PROGRAM DomeControl
VAR_INPUT
	// enable the dome azimuth
	enable:		BOOL;
	// reset the dome axis after an error
	Reset:		BOOL;
	// rotate the dome left (ccw)
	left:		BOOL;
	// rotate the dome right (cw)
	right: 		BOOL;
	// open the dome
	OpenDome:	BOOL;
	// close the dome
	CloseDome:	BOOL; // := TRUE;
	// turn on the light in the dome
	Light: 		BOOL;
	// azimuth position to move to
	position:	LREAL;
	// initiate homing
	HomeAxis:	BOOL;
END_VAR
VAR_OUTPUT
	// error condition on the azimuth drive
	Error:		BOOL;
	// NC axis error of the dome drive
	ErrorID:	UDINT;
	// error in the dome communication or drive
	DomeError:	BOOL;
	// dome is calibrated
	Calibrated:	BOOL;
END_VAR
VAR
	// dome axis function block
	DomeAxis: FB_Axis2;
	// current measured dome azimuth
	Azimuth_current: 	LREAL;
	// dome velocity
	ActVelo:			LREAL;
	//
	//manual_enable:		BOOL;
	// command to move the azimuth to position
	move_azimuth:		BOOL;
	// dome is halted
	//stop_done:			BOOL;
	// dome slit and flap are open
	DomeOpened:			BOOL;
	// dome is closed
	DomeClosed:			BOOL;
	// dome flap (lower section) is open
	FlapOpen:			BOOL;
	// dome flap (lower section) is closed
	FlapClosed:			BOOL;
	//dome slit is open
	SlitOpen:			BOOL;
	// dome slit is closed
	SlitClosed:			BOOL;
	// bit to indicate if domestatus is valid
	DomeValid:			BOOL;
	// dome control word
   	DomeStatusWord:		WORD;
	// last status Word
	LastStatus:			WORD;
	// permanent communication error
	PermanentError:		TON := (IN:=FALSE, PT:=T#30S);
	HomeDelay:			FB_TONTP;
	F_Azimuth_home:		F_TRIG;
	R_Azimuth_home:		R_TRIG;
	// direction invariant azimuth home signal;
	Azimuth_home:		BOOL;
	// time delay for dome light
	LightTimer:			TP;
	// next state
	//:				BYTE := 0;
	// ADS communiaction busy
	bBusy: 				BOOL;
	// ADS communication error
	bError: 			BOOL;
	// ADS communication error id
	nErrID: 			UDINT;
	// cycle timer for the ADS write cycle
	ReadCycle:			TON := (PT:=T#1S);
	
	fbReadReq: ADSREAD := ( NETID := '5.73.45.158.1.1', PORT := 851, TMOUT := DEFAULT_ADS_TIMEOUT );
	DomeCalibration:	MC_SetPosition;
	SyncDome:			BOOL;
	DomeCommEvent:		FB_Eventlog;
	DomeAxisEvent:		FB_Eventlog;
	DomeOpenedEvent:	FB_Eventlog;
	DomeClosedEvent:	FB_Eventlog;
	OpenDomeEvent:		FB_Eventlog;
	CloseDomeEvent:		FB_Eventlog;
	DomeCalibrationEvent: FB_Eventlog;
	MQTTTimer : TON := (PT:=T#10S);
	// MQTT String
	sPayloadPub: STRING(255);
	getlastposition:	BOOL := TRUE;
END_VAR
VAR CONSTANT
	tolerance:				LREAL := 5.0;
	calibration_position:	LREAL := 172.5;
	home_position:			LREAL := 180.0;
END_VAR
VAR PERSISTENT
	last_position:	LREAL := -1.0;
END_VAR

(* This program is responsible for the dome control. 
The dome is enabled unless the emergency button is pressed.
The two-button manual box steers the dome counter-clockwise or clockwise
If the dome is in automatic mode, homing is performed first.
The first section controls the signals for the inverter.
The second section controls the dome axis.
The third section handles the communications via ADS with the dome PLC.
*)

DomeLowLevelControl(enable := GVL_Safety.Run);
enable := GVL_Safety.Run;

// if we are calibrated or encounter an error while calibrating, deactivate homing
IF DomeAxis.Calibrated OR Error THEN
	HomeAxis := FALSE;
END_IF

IF Error THEN
	move_azimuth := FALSE;
END_IF

IF DomeAxis.Calibrated THEN
	last_position := Azimuth_current;
	getlastposition := FALSE;
END_IF


ActVelo := GVL_Dome.ActVelo;

// limit position to sane value
position := MODABS(position, 360.0);

// if we are calibrated, but azimuth is not, go to home position
HomeDelay(IN := DomeAxis.Calibrated, PT1 := T#5S, PT2 := T#100MS);

IF HomeDelay.Q THEN
	position := home_position;
	move_azimuth := TRUE;
END_IF

SyncDome := DomeAxis.Calibrated AND TelescopeControl.power AND AzimuthElevationControl.calibrated;
// if we are on automatic, tie the dome to the telescope

IF DomeAxis.Calibrated AND TelescopeControl.power AND AzimuthElevationControl.calibrated THEN
	position := MODABS(TelescopeControl.azimuth_current, 360.0);
	IF ABS(Azimuth_current - position) > tolerance THEN
		move_azimuth := TRUE;
	ELSE
		move_azimuth := FALSE;
	END_IF
	
END_IF

Calibrated := DomeAxis.Calibrated;
// when homing, ensure that the position is the calibration position
IF HomeAxis THEN
	position := calibration_position;	
END_IF
F_Azimuth_home(CLK := GVL_Dome.Azimut_home);
R_Azimuth_home(CLK := GVL_Dome.Azimut_home);

Azimuth_home := (R_Azimuth_home.Q AND GVL_Dome.bDirectionPlus) OR 
				(F_Azimuth_home.Q AND GVL_Dome.bDirectionMinus);

// velocity = 2°/s or 180° in 81s, 360° in 120s (was 2.22)
// TODO: Reset does not propagate to the FB and therefor does not reset the error
DomeAxis(
	Enable := 		enable,
	Reset := 		reset,
	MoveAxis := 	move_azimuth,
	HomeAxis :=		HomeAxis,
	Position := 	position,
	Velocity := 	3.0,
	Jog_Forward :=	right OR GVL_Dome.Clockwise,
	Jog_Backwards := left OR GVL_Dome.CounterClockwise,
	bCalibrationCam := GVL_Dome.Azimut_home,
	isModuloAxis := TRUE,
	//StopDone =>		stop_done,
	Error =>		error,
	ErrorID =>		ErrorID,
	ActualPosition => Azimuth_current,
	AxisRef	:= 		GVL_Dome.DomeAxisRef);

IF getlastposition AND last_position>=0.0 AND NOT Calibrated THEN
	DomeCalibration.Execute := getlastposition AND DomeAxis.Ready;
	DomeCalibration.Position := last_position;
ELSE
	DomeCalibration.Execute := Azimuth_home AND HomeDelay.Q AND DomeAxis.Ready;
	DomeCalibration.Position := calibration_position;
END_IF

// re-calibrate the dome, if we pass the reference switch. execute only if enough time has passed since homing.
DomeCalibration(Axis := GVL_Dome.DomeAxisRef);

IF DomeCalibration.Done OR Calibrated THEN
	getlastposition := FALSE;
END_IF

IF DomeAxis.MoveDone THEN
	move_azimuth := FALSE;
END_IF


// Light is switched off after 60 minutes or if Light signal is low
LightTimer(IN := Light, PT := T#60M);
GVL_Dome.Light := Light AND LightTimer.Q;

(* The remote section for moving parts of the dome starts here. *)
GVL_Dome.DomeControlWord.0 := TRUE;
IF CloseDome THEN
	OpenDome := FALSE;
	GVL_Dome.DomeControlWord.1 := TRUE; // CloseFlap
	GVL_Dome.DomeControlWord.2 := TRUE; // CloseSlit
	GVL_Dome.DomeControlWord.3 := FALSE; // OpenFlap
	GVL_Dome.DomeControlWord.4 := FALSE; // OpenSlit
ELSIF OpenDome THEN
	GVL_Dome.DomeControlWord.1 := FALSE; // CloseFlap
	GVL_Dome.DomeControlWord.2 := FALSE; // CloseSlit
	GVL_Dome.DomeControlWord.3 := TRUE; // OpenFlap
	GVL_Dome.DomeControlWord.4 := TRUE; // OpenSlit
ELSE
	GVL_Dome.DomeControlWord.1 := FALSE; // CloseFlap
	GVL_Dome.DomeControlWord.2 := FALSE; // CloseSlit
	GVL_Dome.DomeControlWord.3 := FALSE; // OpenFlap
	GVL_Dome.DomeControlWord.4 := FALSE; // OpenSlit
END_IF

ReadCycle(IN := TRUE);
IF ReadCycle.Q THEN
	// read if the ADS command is busy
	fbReadReq(	READ := FALSE,
				BUSY => bBusy,
				ERR =>	bError,
				ERRID => nErrID);
	IF bBusy THEN
		// reset the read command
		fbReadReq(READ := FALSE);
	ELSE
		// read the variable
		fbReadReq(  IDXGRP := 16#4020, 
					IDXOFFS := 0, 
					LEN := SIZEOF(DomeStatusWord), 
					DESTADDR := ADR(DomeStatusWord),
					READ := TRUE,
					BUSY => bBusy,
					ERR =>	bError,
					ERRID => nErrID);
		// restart the read cycle
		ReadCycle(IN := FALSE);		
	END_IF
	
	IF NOT bError THEN
		DomeValid  := DomeStatusWord.0;
		DomeOpened := DomeStatusWord.1;
		DomeClosed := DomeStatusWord.2;
		FlapOpen   := DomeStatusWord.3;
		FlapClosed := DomeStatusWord.4;
		SlitOpen   := DomeStatusWord.5;
		SlitClosed := DomeStatusWord.6;
	ELSE
		// reset the status word
		DomeStatusWord := 0;
	END_IF
END_IF

CASE NErrID OF
			6: DomeCommEvent.OnMessage := 'ERR_TARGETPORTNOTFOUND';
			29: DomeCommEvent.OnMessage := 'ERR_AMSSYNC_TIMEOUT';
			1861: DomeCommEvent.OnMessage := 'ADSERR_CLIENT_SYNCTIMEOUT';
ELSE
			DomeCommEvent.OnMessage := UDINT_TO_STRING(nErrID);
END_CASE

PermanentError(IN := bError);
		
DomeError := PermanentError.Q OR Error;

IF DomeOpened THEN
	OpenDome := FALSE;
ELSIF DomeClosed THEN
	CloseDome := FALSE;
END_IF

MQTTTimer(IN:=Enable);
IF MQTTTimer.Q THEN // publish new payload every second
	MQTTTimer(IN:=FALSE);
	sPayloadPub := 'dome,location=dome,host=CX-4E6032 ';
	sPayloadPub := APPEND(sPayloadPub, 'DomeAzimuth=', LREAL_TO_FMTSTR(Azimuth_current, 1, TRUE));
	sPayloadPub := APPEND(sPayloadPub, ',Calibrated=', BOOL_TO_STRING(Calibrated));	
	MQTTCommunication.fbMqttClient.Publish(	
					sTopic:= 'RoboTel/Telemetry', 
					pPayload:= ADR(sPayloadPub), 
					nPayloadSize:= LEN2(ADR(sPayloadPub)),
					eQoS:= TcIotMqttQos.AtMostOnceDelivery,
					bRetain:= FALSE, 
					bQueue:= FALSE );
	// invalidate last status for testing
	LastStatus := 0;
END_IF

IF DomeStatusWord <> LastStatus THEN
	LastStatus := DomeStatusWord;
	sPayloadPub := 'dome,location=dome,host=CX-4E6032,module=DomeControl ';
	sPayloadPub := APPEND(sPayloadPub, 'DomeCommunicationOK=', BOOL_TO_STRING(NOT PermanentError.Q));
	sPayloadPub := APPEND(sPayloadPub, ',DomeClosed=', BOOL_TO_STRING(DomeClosed));
	sPayloadPub := APPEND(sPayloadPub, ',DomeOpened=', BOOL_TO_STRING(DomeOpened));
	sPayloadPub := APPEND(sPayloadPub, ',FlapOpen=', BOOL_TO_STRING(FlapOpen));	
	sPayloadPub := APPEND(sPayloadPub, ',FlapClosed=', BOOL_TO_STRING(FlapClosed));	
	sPayloadPub := APPEND(sPayloadPub, ',SlitOpen=', BOOL_TO_STRING(SlitOpen));	
	sPayloadPub := APPEND(sPayloadPub, ',SlitClosed=', BOOL_TO_STRING(SlitClosed));	
	
	MQTTCommunication.fbMqttClient.Publish(	
					sTopic:= 'RoboTel/Telemetry', 
					pPayload:= ADR(sPayloadPub), 
					nPayloadSize:= LEN2(ADR(sPayloadPub)),
					eQoS:= TcIotMqttQos.AtMostOnceDelivery,
					bRetain:= TRUE, 
					bQueue:= FALSE );
END_IF

DomeCommEvent(	Trigger := PermanentError.Q, 
					Level := ADSLOG_MSGTYPE_ERROR,
					FormatString := 'Dome communication error: %s',
					OffMessage := 'OK',
					OffLevel := ADSLOG_MSGTYPE_HINT);
DomeAxisEvent(	
	Trigger := 		Error, 
	Level := 		ADSLOG_MSGTYPE_ERROR,
	FormatString :=	'Dome axis Error: %s',
	OnMessage := 	NCError_TO_STRING(ErrorID),
	OffMEssage := 	'OK');
				
DomeCalibrationEvent(	
	Trigger := 		GVL_Dome.Azimut_home, 
	Level := 		ADSLOG_MSGTYPE_HINT,
	OnMessage := 	'Dome is (re-)calibrated.');

DomeOpenedEvent(
	Trigger := 		DomeOpened, 
	Level := 		ADSLOG_MSGTYPE_WARN,
	OnMessage := 	'Dome is open.');
	
DomeClosedEvent(
	Trigger := 		DomeClosed, 
	Level := 		ADSLOG_MSGTYPE_HINT,
	OnMessage := 	'Dome is closed.');
	
OpenDomeEvent(
	Trigger := 		OpenDome, 
	Level := 		ADSLOG_MSGTYPE_WARN,
	OnMessage := 	'Dome is opening.');
	
CloseDomeEvent(
	Trigger := 		CloseDome, 
	Level := 		ADSLOG_MSGTYPE_HINT,
	OnMessage := 	'Dome is closing.');

END_PROGRAM

(* stored: Version 1.1.0.1, ProductVersion 3.1.4024.9
   POU DomeControl: Id {0e02434d-920e-4c0f-81fc-5ff7d5573875}, SpecialFunc None *)
